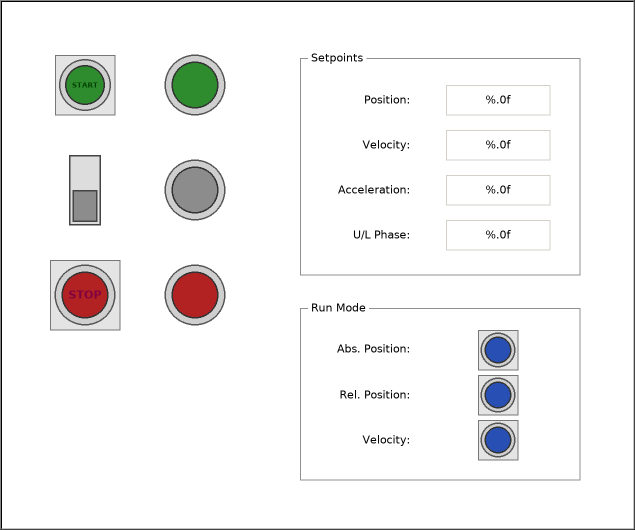
VISUALIZATION hmi  // 635x530
    RoundedRectangle (0,0 635x530)
    PushSwitch (55,55 60x60), tooltip "START", variable: MAIN.togStart, behaviour: TOGGLE, style: Switch-PushSwitch-Green
    Lamp1 (160,50 70x70), variable: MAIN.togStart, style: Lamp-Lamp1-Green
    PushSwitch (50,260 70x70), tooltip "STOP", variable: MAIN.togStop, behaviour: TOGGLE, style: Switch-PushSwitch-Red
    Lamp1 (160,260 70x70), variable: MAIN.togStop, style: Lamp-Lamp1-Red
    GroupBox (300,50 280x225), "Setpoints"
        Label (16,80 97x30), "Velocity:"
        Label (16,125 97x30), "Acceleration:"
        Textfield (146,80 104x30), "%.0f", text variable: MAIN.txtVel
            OnMouseClick: write the text variable via InputWithLimits, format %d
        Textfield (146,35 104x30), "%.0f", text variable: MAIN.txtPos
            OnMouseClick: write the text variable via InputWithLimits
            OnMouseClick: change screen: 
        Textfield (146,125 104x30), "%.0f", text variable: MAIN.txtAcc
            OnMouseClick: write the text variable via InputWithLimits, format %d
        Label (16,35 97x30), "Position:"
        Label (16,170 97x30), "U/L Phase:"
        Textfield (146,170 104x30), "%.0f", text variable: MAIN.txtPhs
            OnMouseClick: write the text variable via InputWithLimits, format %d
    GroupBox (300,300 280x180), "Run Mode"
        Label (16,80 97x30), "Rel. Position:"
        Label (16,125 97x30), "Velocity:"
        Label (16,34 97x30), "Abs. Position:"
        PushSwitch (178,30 40x40), variable: MAIN.togAbsPos, behaviour: TOGGLE, style: Switch-PushSwitch-Blue
        PushSwitch (178,75 40x40), variable: MAIN.togRelPos, behaviour: TOGGLE, style: Switch-PushSwitch-Blue
        PushSwitch (178,120 40x40), variable: MAIN.togVel, behaviour: TOGGLE, style: Switch-PushSwitch-Blue
    DipSwitch (50,155 70x70), tooltip "COUPLE", variable: MAIN.togCoup, behaviour: TOGGLE, style: Switch-DipSwitch-Gray
    Lamp1 (160,155 70x70), variable: MAIN.togCoup, style: Lamp-Lamp1-Gray
    Label (60,280 50x30), "STOP"
    Label (60,70 50x30), "START"
END_VISUALIZATION

(* stored: Version 1.1.0.1, ProductVersion 3.1.4024.12
   Visu hmi: Id {871559c6-b0ee-4414-8ee3-84a32fbb96ef} *)
